// LS Electric XG5000 project: 8_29_문제3
// PLC LSPLC

PROGRAM NewProgram (task: 스캔 프로그램)

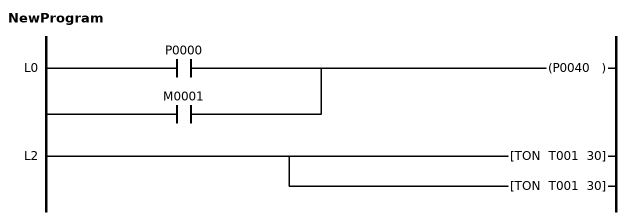
; L0
LOAD      P0000
OR        M0001
OUT       P0040
; L2
TON       T001 30
TON       T001 30